(*
This file is present, but not yet tracked in the PLC project file.
*)
FUNCTION F_UntrackedFunc : BOOL
VAR_INPUT
END_VAR
VAR
END_VAR

F_UntrackedFunc := TRUE;

END_FUNCTION

(* stored: Version 1.1.0.1, ProductVersion 3.1.4024.11
   POU F_UntrackedFunc: Id {9722563b-e568-4fd9-9af1-e72780fe078b}, SpecialFunc None *)
